RoboDK station: robodk_cube_workstation.rdk

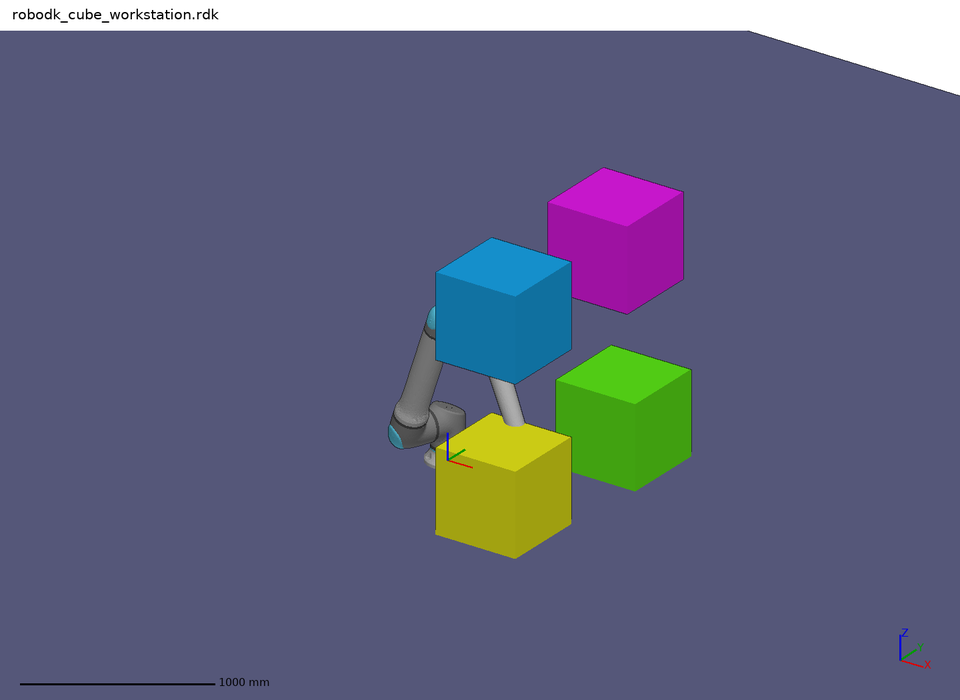
[picture v0: the station drawn from its stored meshes, robots at their saved joint values, targets as dots, program paths as lines]
Station New Station (1) (saved by RoboDK 5.2.4). Poses are relative to the parent item; angles as X-Y-Z fixed-axis rotations.
  - frame UR20 Base at (0, 0, 0) mm
    - robot UR20: 6 axes
        modified DH rows (alpha deg, a mm, theta deg, d mm): 0, 0, 0, 236.2; 90, 0, -180, 0; 0, 861.8, 0, 0; 0, 727.7, 0, 201.9; -90, 0, 0, 159.4; 90, 0, 0, 154.8
        joint limits [-360, -360, -360, -360, -360, -360] to [360, 360, 360, 360, 360, 360]; home [0, -90, -90, 0, 90, 0]; saved at [-20.606, -113.195, -124.795, -34.395, 89.199, -20.589]
    - item type 7 baselight_1
    - item type 7 baselight_2
  - object plane at (0, 0, 0) mm, size 10000 x 10000 x 0 mm, geometry from plane.obj
  - object cube at (750, 500, 0) mm, size 500 x 500 x 500 mm, geometry from cube.obj
  - object cube at (700, -500, 0) mm, size 500 x 500 x 500 mm, geometry from cube.obj
  - object cube at (700, 500, 1000) mm, size 500 x 500 x 500 mm, geometry from cube.obj
  - object cube at (700, -500, 1000) mm, size 500 x 500 x 500 mm, geometry from cube.obj
